FUNCTION ATAN2 : LREAL
VAR_INPUT
	y, x: LREAL;
END_VAR
VAR
END_VAR

(* source: https://de.wikipedia.org/wiki/Arctan2 *)
ATAN2 := 0.0;

IF x > 0 THEN
	ATAN2 := ATAN(y/x);
ELSIF x < 0 AND y > 0 THEN
	ATAN2 := ATAN(y/x) + PI;
ELSIF x < 0 AND y = 0 THEN
	ATAN2 := PI;
ELSIF x < 0 AND y < 0 THEN
	ATAN2 := ATAN(y/x) - PI;
ELSIF x = 0 AND y > 0 THEN
	ATAN2 := PI/2.0;
ELSIF x = 0 AND y < 0 THEN
	ATAN2 := -PI/2.0;
END_IF

END_FUNCTION

(* stored: Version 1.1.0.1, ProductVersion 3.1.4024.9
   POU ATAN2: Id {dba69bd6-0eda-4092-a354-7cdf0084c954}, SpecialFunc None *)
